KUKA KRL program: KUKA_robot.src

&ACCESS RV
&PARAM TEMPLATE C:\KRC\Roboter\Template\vorgabe
&PARAM EDITMASK

DEF test()

   FOLD INI
      FOLD BASISTECH INI
         GLOBAL INTERRUPT DECL 3 WHEN SSTOPMESS == TRUE DO IR_STOPM()
         INTERRUPT ON 3
         BAS (#INITMOV, 0)
      ENDFOLD (BASISTECH INI)

      FOLD USER INI
         ; Make your modifications here
      ENDFOLD (USER INI)
   ENDFOLD (INI)

   FOLD PTP HOME Vel=100% DEFAULT ; %[PE]SMKUKATPBASIS, SCMOVE, %VPTP, %P 1:PTP, 2: HOME, 3, 5:100, 7: DEFAULT
      SBWDSTART = FALSE
      PDAT_ACT = PDEFAULT
      FDAT_ACT = FHOME
      BAS (#PTP_PARAMS, 100)
      PTP XHOME
   ENDFOLD

   LOOP
      FOLD PTP P1 Vel=100% PDAT1 Tool[1] Base[0]; %[PE]SMKUKATPBASIS, SCMOVE, %VPTP, %P 1:PTP, 2:P1, 3, 5:100, 7:PDAT1
         SBWDSTART = FALSE
         PDAT_ACT = PPDAT1
         FDAT_ACT = FP1
         BAS (#PTP_PARAMS, 100)
         PTP P1
      ENDFOLD

      ; Additional movements or logic can be added here
      ; Example:
      PTP P2
      PTP P3
      PTP P4
   ENDLOOP

END
